PROGRAM Socket
VAR
	arSocketListen: ARRAY[1..8] OF FB_SocketListen;
	arSocketAccept: ARRAY[1..8] OF FB_SocketAccept;	
	
	arSocketConnect: ARRAY[1..8] OF FB_SocketConnect;
	arSocketReceive: ARRAY[1..8] OF FB_SocketReceive;
    arSocketSend: ARRAY[1..8] OF FB_SocketSend;	
	arSocketClose: ARRAY[1..8] OF FB_SocketClose;	
		
	arListen: ARRAY[1..8] OF BOOL;
	arhlistener: ARRAY[1..8] OF  T_HSOCKET;

	wReceiveDataBuffer: ARRAY[0..127] OF WORD;
	wSendDataBuffer: ARRAY[0..127] OF WORD;	
	
	wReceiveData: ARRAY[0..127] OF WORD;
	wSendData: ARRAY[0..127] OF WORD;
	wNullData: ARRAY[0..127] OF WORD;
	
	pbyReceiveData: ARRAY [0..255] OF BYTE;;
	pbySendData: ARRAY [0..255] OF BYTE;;
 
	byReceiveData: ARRAY [0..255] OF BYTE;;
	bySendData: ARRAY [0..255] OF BYTE;	
	
	byPrint:  ARRAY [0..MAX_STRING_LENGTH] OF BYTE;
	byPrintAuto:  ARRAY [0..MAX_STRING_LENGTH] OF BYTE;
	byPrintUser:  ARRAY [0..MAX_STRING_LENGTH] OF BYTE;
	
	iSocket: ARRAY[1..8] OF INT;
	arConnectExecute: ARRAY[1..8] OF BOOL;
	arConnectError: ARRAY[1..8] OF BOOL;
	arConnectErrId: ARRAY[1..8] OF UDINT;
	arConnectBusy: ARRAY[1..8] OF BOOL;
		
	arReceiveExecute: ARRAY[1..8] OF BOOL;
	arReceiveError: ARRAY[1..8] OF BOOL;
	arReceiveErrId: ARRAY[1..8] OF UDINT;
	arReceiveBusy: ARRAY[1..8] OF BOOL;
		
	arCloseExecute: ARRAY[1..8] OF BOOL;
	arCloseError: ARRAY[1..8] OF BOOL;
	arCloseErrId: ARRAY[1..8] OF UDINT;
	arCloseBusy: ARRAY[1..8] OF BOOL;
	arhSocket: ARRAY[1..8] OF T_HSOCKET;
	
	arSendExecute: ARRAY[1..8] OF BOOL;

	
	arSendError: ARRAY[1..8] OF BOOL;
	arSendErrId: ARRAY[1..8] OF UDINT;
	arSendBusy: ARRAY[1..8] OF BOOL;
	arTon: ARRAY [1..8] OF Ton;
	arBlink: ARRAY[1..8] OF BLINK;
	
	testString: STRING:='1';
	byteString: BYTE;
	pS: POINTER TO STRING;

	arAccept: ARRAY[1..8] OF bool;
	arListenBusy: ARRAY[1..8] OF bool;
	arAcceptBusy: ARRAY[1..8] OF bool;
	arListenError: ARRAY[1..8] OF bool;
	arAcceptError: ARRAY[1..8] OF bool;

	
	
	byPrintSend: ARRAY [0..MAX_STRING_LENGTH] OF BYTE;
	byPrintReceive: ARRAY [0..MAX_STRING_LENGTH] OF BYTE;


	iPPReceive: INT;
	diReceiveData: DINT;
	iPPSend: INT;
	iPPAccept: INT;

	
	tonFS: TON;
	
	pReceiveString: POINTER TO STRING;
	wSendCnt: WORD;
	
	
	sTestSting: STRING(255);
	arrtestBytearr: ARRAY [0..MAX_STRING_LENGTH] OF BYTE;
	arrToBytearr: ARRAY [0..MAX_STRING_LENGTH] OF BYTE;
	sToBytearrString: T_MaxString;
	sAutoPrintData: STRING(22);
	sTestPrintData: STRING(22);
	bDebugFlag: DINT;
	sTestData: STRING;
	iLen: UINT;
	rViewPrintPos: REAL;
	rPrintPosBuffer: REAL;
END_VAR

//TCP1_Client();
TCP2_Server();
pReceiveString:=ADR(pbyReceiveData);
HMI_PrinterReceiveData:=pReceiveString^;
sTestSting:=BYTEARR_TO_MAXSTRING(in:= arrtestBytearr);
arrToBytearr:=MAXSTRING_TO_BYTEARR(in:= sToBytearrString);

ACTION TCP1_Client:
(*
arSocketConnect[1](
	sSrvNetId:= , 
	sRemoteHost:= '192.168.1.199', 
	nRemotePort:= 3000, 
	bExecute:= arConnectExecute[1] , 
	tTimeout:= T#10S, 
	bBusy=> arConnectBusy[1], 
	bError=> arConnectError[1], 
	nErrId=> arConnectErrId[1], 
	hSocket=> arhSocket[1]);
		
arBlink[1](TimeH:= 1000, TimeL:= 2000, OUT=> );
	
arSocketReceive[1](
	sSrvNetId:= , 
	hSocket:=  arhSocket[1], 
	cbLen:= 255, 
	pDest:= ADR(ReceiveData[1]), 
	bExecute:= arReceiveExecute[1], 
	tTimeout:= T#1S, 
	bBusy=> arReceiveBusy[1], 
	bError=> arReceiveError[1], 
	nErrId=> arReceiveErrId[1], 
	nRecBytes=> );

arSocketSend[1](
	sSrvNetId:= , 
	hSocket:= arhSocket[1], 
	cbLen:=  255, 
	pSrc:= ADR(SendData[1]), 
	bExecute:= arSendExecute[1], 
	tTimeout:= T#1S, 
	bBusy=> arSendBusy[1], 
	bError=> arSendError[1], 
	nErrId=> arSendErrId[1]);	
	
	
arSocketClose[1](
	sSrvNetId:= , 
	hSocket:=  arhSocket[1], 
	bExecute:= arCloseExecute[1], 
	tTimeout:= T#1S, 
	bBusy=>  arCloseBusy[1], 
	bError=> arCloseError[1], 
	nErrId=> arCloseErrId[1]);



	
CASE iSocket[1] OF 
0:  
    MEMSET(destAddr:= ADR(arhSocket[1]), fillByte:= 0, n:= SIZEOF(arhSocket[1]));  
	arConnectExecute[1]:=FALSE;	
    iSocket[1]:=1;
	
1:  
	iSocket[1]:=2;
		
2:
    arConnectExecute[1]:=TRUE;	
    IF arConnectBusy[1] THEN
	   arConnectExecute[1]:=FALSE;	
       iSocket[1]:=3;
	END_IF	
	
3:  
	iSocket[1]:=4;
	
4:	
    IF arhSocket[1].handle<>0 THEN
       iSocket[1]:=10;
	ELSE IF arConnectError[1] THEN
		    iSocket[1]:=0;
		 END_IF
	END_IF


	   
10:
    arReceiveExecute[1]:=TRUE;
	iSocket[1]:=11;
	
11:
	   arReceiveExecute[1]:=FALSE;
	   iSocket[1]:=12;
12:
	IF NOT arReceiveError[1] AND NOT arReceiveBusy[1] THEN
	   iSocket[1]:=13;
	   ELSE IF arReceiveError[1] THEN
	           iSocket[1]:=90; 
            END_IF  
	END_IF 	
	
13:	
	   iSocket[1]:=20;
	
20:
	arSendExecute[1]:=TRUE; 
	iSocket[1]:=21;


21:	 
	   arSendExecute[1]:=FALSE;
	   iSocket[1]:=22;
	
22:
	IF NOT arSendError[1] AND NOT arSendBusy[1]  THEN
	   iSocket[1]:=23;
	   ELSE IF arSendError[1] THEN
	           iSocket[1]:=90;
	        END_IF
	END_IF 
       		   
23:
	   iSocket[1]:=10;


90: 
    arConnectExecute[1]:=FALSE;  
    arSendExecute[1]:=FALSE;
    arReceiveExecute[1]:=FALSE;
	arCloseExecute[1]:=TRUE;
	iSocket[1]:=91;

91: 
	   iSocket[1]:=92;

92:
	   arCloseExecute[1]:=FALSE;
	   iSocket[1]:=0;

END_CASE
*)
END_ACTION

ACTION TCP2_Server:
tonFS(IN:= TRUE, PT:= T#60S, Q=> , ET=> );

arSocketListen[2](
	sSrvNetId:= , 
	sLocalHost:= '192.168.1.10', 
	nLocalPort:= 6853, 
	bExecute:= arListen[2] OR tonFS.Q , 
	tTimeout:=, 
	bBusy=> arListenBusy[2], 
	bError=> arListenError[2], 
	nErrId=> , 
	hListener=> arhlistener[2]);
	
	
arSocketAccept[2](
	sSrvNetId:= , 
	hListener:= arhlistener[2], 
	bExecute:= arAccept[2], 
	tTimeout:= , 
	bAccepted=> , 
	bBusy=> arAcceptBusy[2], 
	bError=> arAcceptError[2], 
	nErrId=> , 
	hSocket=> arhSocket[2]);	
	
arSocketReceive[2](
	sSrvNetId:= , 
	hSocket:=  arhSocket[2], 
	cbLen:= 255, 
	pDest:= ADR(wReceiveDataBuffer), 
	bExecute:= arReceiveExecute[2], 
	tTimeout:= T#1S, 
	bBusy=> arReceiveBusy[2], 
	bError=> arReceiveError[2], 
	nErrId=> arReceiveErrId[2], 
	nRecBytes=> );

arSocketSend[2](
	sSrvNetId:= , 
	hSocket:= arhSocket[2], 
	cbLen:=  255, 
	pSrc:= ADR(wSendDataBuffer), 
	bExecute:= arSendExecute[2], 
	tTimeout:= T#1S, 
	bBusy=> arSendBusy[2], 
	bError=> arSendError[2], 
	nErrId=> arSendErrId[2]);	
	
	
arSocketClose[2](
	sSrvNetId:= , 
	hSocket:=  arhSocket[2], 
	bExecute:= arCloseExecute[2], 
	tTimeout:= T#1S, 
	bBusy=>  arCloseBusy[2], 
	bError=> arCloseError[2], 
	nErrId=> arCloseErrId[2]);	
	
	
rViewPrintPos:= arRealAxisAdmin[48].o.ActPos- rPrintPosBuffer;
	
CASE iPPAccept OF 
0:  
    MEMSET(destAddr:= ADR(wReceiveData), fillByte:= 0, n:= SIZEOF(wReceiveData));
    MEMSET(destAddr:= ADR(arhSocket[2]), fillByte:= 0, n:= SIZEOF(arhSocket[2]));  		
    iPPAccept:=1;	
1: 	
    IF arhlistener[2].handle<>0 THEN
       iPPAccept:=2;
	END_IF
2:	
	arTon[2](IN:= TRUE, PT:= T#100MS, Q=> , ET=> );	
	IF arTon[2].Q THEN
	   arTon[2](IN:= FALSE, PT:= T#100MS, Q=> , ET=> );	
	   iPPAccept:=10;
	END_IF
	   
10: arAccept[2]:=TRUE;	
    iPPAccept:=11;
	
11:
	arTon[2](IN:= TRUE, PT:= T#100MS, Q=> , ET=> );	
	IF arTon[2].Q THEN
	   arTon[2](IN:= FALSE, PT:= T#100MS, Q=> , ET=> );	
	   iPPAccept:=12;
	END_IF
	
12:	
    IF arhSocket[2].handle<>0 THEN
       iPPAccept:=20;
	   ELSE 
	   arAccept[2]:=FALSE;
	   iPPAccept:=1;
	END_IF

20:
    HMI_PrinterConnected:=TRUE;
    iPPReceive:=10;
	iPPAccept:=100;


90:  
    
    HMI_PrinterConnected:=FALSE;
	arAccept[2]:=FALSE;
    arSendExecute[2]:=FALSE;
    arReceiveExecute[2]:=FALSE;
	arCloseExecute[2]:=TRUE;
	iPPAccept:=91;

91: 
	arTon[2](IN:= TRUE, PT:= T#100MS, Q=> , ET=> );	
	IF arTon[2].Q THEN
	   arTon[2](IN:= FALSE, PT:= T#100MS, Q=> , ET=> );	
	   iPPAccept:=92;
	END_IF
	
92:
	arCloseExecute[2]:=FALSE;
	iPPAccept:=0;
END_CASE
	
CASE iPPReceive OF
	10: 
	    MEMSET(destAddr:= ADR(wReceiveDataBuffer), fillByte:= 0, n:= SIZEOF(wReceiveDataBuffer));
	    arReceiveExecute[2]:=FALSE;
		iPPReceive:=11;
		
	11:
        arTon[3](IN:= TRUE, PT:= T#100MS, Q=> , ET=> );	
		IF arTon[3].Q THEN
		   arTon[3](IN:= FALSE, PT:= T#100MS, Q=> , ET=> );	
		   iPPReceive:=20;
		END_IF
		
	20:	
	    arReceiveExecute[2]:=TRUE;
		iPPReceive:=21;
		
	21:
        arTon[3](IN:= TRUE, PT:= T#1000MS, Q=> , ET=> );	
		IF arTon[3].Q THEN
		   arTon[3](IN:= FALSE, PT:= T#1000MS, Q=> , ET=> );	
		   iPPReceive:=30;
		END_IF		
		
	30: 
        diReceiveData:=MEMCMP(pBuf1:=ADR(wReceiveDataBuffer) , pBuf2:=ADR(wNullData) , n:=SIZEOF(wNullData));
        IF 	diReceiveData<>0 THEN
		    MEMSET(destAddr:= ADR(wReceiveData), fillByte:= 0, n:= SIZEOF(wReceiveData));
		    wReceiveData:=wReceiveDataBuffer;
			pbyReceiveData[0]:=WORD_TO_BYTE(wReceiveDataBuffer[5]);
			pbyReceiveData[1]:=WORD_TO_BYTE(wReceiveDataBuffer[6]);
			pbyReceiveData[2]:=WORD_TO_BYTE(wReceiveDataBuffer[7]);
			pbyReceiveData[3]:=WORD_TO_BYTE(wReceiveDataBuffer[8]);
			pbyReceiveData[4]:=WORD_TO_BYTE(wReceiveDataBuffer[9]);
			pbyReceiveData[5]:=WORD_TO_BYTE(wReceiveDataBuffer[10]);
			pbyReceiveData[6]:=WORD_TO_BYTE(wReceiveDataBuffer[11]);
			pbyReceiveData[7]:=WORD_TO_BYTE(wReceiveDataBuffer[12]);
			pbyReceiveData[8]:=WORD_TO_BYTE(wReceiveDataBuffer[13]);
			pbyReceiveData[9]:=WORD_TO_BYTE(wReceiveDataBuffer[14]);
			pbyReceiveData[10]:=WORD_TO_BYTE(wReceiveDataBuffer[15]);
			pbyReceiveData[11]:=WORD_TO_BYTE(wReceiveDataBuffer[16]);
			pbyReceiveData[12]:=WORD_TO_BYTE(wReceiveDataBuffer[17]);
			pbyReceiveData[13]:=WORD_TO_BYTE(wReceiveDataBuffer[18]);
			pbyReceiveData[14]:=WORD_TO_BYTE(wReceiveDataBuffer[19]);
			pbyReceiveData[15]:=WORD_TO_BYTE(wReceiveDataBuffer[20]);
			pbyReceiveData[16]:=WORD_TO_BYTE(wReceiveDataBuffer[21]);
			pbyReceiveData[17]:=WORD_TO_BYTE(wReceiveDataBuffer[22]);
			pbyReceiveData[18]:=WORD_TO_BYTE(wReceiveDataBuffer[23]);
			pbyReceiveData[19]:=WORD_TO_BYTE(wReceiveDataBuffer[24]);
			pbyReceiveData[20]:=WORD_TO_BYTE(wReceiveDataBuffer[25]);
			pbyReceiveData[21]:=WORD_TO_BYTE(wReceiveDataBuffer[26]);
			pbyReceiveData[22]:=WORD_TO_BYTE(wReceiveDataBuffer[27]);			
	    END_IF
		iPPReceive:=10;
	    IF arSocketReceive[2].bError THEN
		   iPPReceive:=0;
		   iPPAccept:=90;
		END_IF
		
END_CASE

CASE iPPSend OF
	0:  IF HMI_PrinterConnected  AND glb_Un02Box.Box[HMI_PrintNo].PrintRequest AND wReceiveData[0]<>0 THEN
		   iPPSend:=10;
		ELSE IF HMI_PrinterConnected AND wReceiveData[0]<>0 AND  HMI_PrinterTest THEN
                iPPSend:=200;
			 END_IF	
	    END_IF
	10:
	   MEMSET(destAddr:= ADR(byPrintUser), fillByte:= 0, n:= SIZEOF(byPrintUser));
	   MEMSET(destAddr:= ADR(wSendDataBuffer), fillByte:= 0, n:= SIZEOF(wSendDataBuffer));
	   MEMSET(destAddr:= ADR(sAutoPrintData), fillByte:= 0, n:= SIZEOF(sAutoPrintData));
	   iLen:=INT_TO_UINT(LEN(glb_Un02Box.Box[HMI_PrintNo].PrintData));
	   MEMCPY(ADR(sAutoPrintData),ADR(glb_Un02Box.Box[HMI_PrintNo].PrintData),ilen);
	   IF NOT bDebugFlag.0 THEN
	   iPPSend:=11;
	   END_IF
	11:
	   byPrintUser:=MAXSTRING_TO_BYTEARR(sAutoPrintData);
	   IF NOT bDebugFlag.1 THEN
	   iPPSend:=20;
       END_IF
	
	   
	20:		
        wSendDataBuffer[0]:= 35;
		iPPSend:=30;
	30: 	
	    wSendCnt:=wSendCnt+1;
	    IF wSendCnt>200 THEN
		   wSendCnt:=1;
		END_IF	
		
		wSendDataBuffer[1]:=0;
		wSendDataBuffer[2]:=wSendCnt;
		wSendDataBuffer[3]:=0;
		wSendDataBuffer[4]:=44;
		wSendDataBuffer[5]:=BYTE_TO_WORD(byPrintUser[0]);
		wSendDataBuffer[6]:=BYTE_TO_WORD(byPrintUser[1]);
		wSendDataBuffer[7]:=BYTE_TO_WORD(byPrintUser[2]);
		wSendDataBuffer[8]:=BYTE_TO_WORD(byPrintUser[3]);
		wSendDataBuffer[9]:=BYTE_TO_WORD(byPrintUser[4]);
		wSendDataBuffer[10]:=BYTE_TO_WORD(byPrintUser[5]);
		wSendDataBuffer[11]:=BYTE_TO_WORD(byPrintUser[6]);
		wSendDataBuffer[12]:=BYTE_TO_WORD(byPrintUser[7]);
		wSendDataBuffer[13]:=BYTE_TO_WORD(byPrintUser[8]);
		wSendDataBuffer[14]:=BYTE_TO_WORD(byPrintUser[9]);
		wSendDataBuffer[15]:=BYTE_TO_WORD(byPrintUser[10]);
		wSendDataBuffer[16]:=BYTE_TO_WORD(byPrintUser[11]);
		wSendDataBuffer[17]:=BYTE_TO_WORD(byPrintUser[12]);
		wSendDataBuffer[18]:=BYTE_TO_WORD(byPrintUser[13]);
		wSendDataBuffer[19]:=BYTE_TO_WORD(byPrintUser[14]);
		wSendDataBuffer[20]:=BYTE_TO_WORD(byPrintUser[15]);
		wSendDataBuffer[21]:=BYTE_TO_WORD(byPrintUser[16]);
		wSendDataBuffer[22]:=BYTE_TO_WORD(byPrintUser[17]);
		wSendDataBuffer[23]:=BYTE_TO_WORD(byPrintUser[18]);
		wSendDataBuffer[24]:=BYTE_TO_WORD(byPrintUser[19]);
		wSendDataBuffer[25]:=BYTE_TO_WORD(byPrintUser[20]);
        wSendDataBuffer[26]:=BYTE_TO_WORD(byPrintUser[21]);	
		arSendExecute[2]:=FALSE;		
		iPPSend:=31;
		
		
    31:		
	    arTon[4](IN:= TRUE, PT:= T#100MS, Q=> , ET=> );	
		IF arTon[4].Q THEN
		   arTon[4](IN:= FALSE, PT:= T#100MS, Q=> , ET=> );	
		   iPPSend:=40;
		END_IF	
    40:
        arSendExecute[2]:=TRUE;
		iPPSend:=41;	
    41:
	    arTon[4](IN:= TRUE, PT:= T#10S, Q=> , ET=> );	
		IF arTon[4].Q THEN
		   arTon[4](IN:= FALSE, PT:= T#10S, Q=> , ET=> );	
		   iPPSend:=50;
		END_IF
		
	50:	
	    arTon[4](IN:= TRUE, PT:= DINT_TO_TIME(HMI_PrintMaxTime*1000), Q=> , ET=> );	
	    IF wReceiveData[2]=wSendCnt  THEN
		   arTon[4](IN:= FALSE, PT:= DINT_TO_TIME(HMI_PrintMaxTime*1000), Q=> , ET=> );
		   iPPSend:=60;
		   ELSE IF arTon[4].Q THEN
				   arTon[4](IN:= FALSE, PT:= DINT_TO_TIME(HMI_PrintMaxTime*1000), Q=> , ET=> );
				   iPPSend:=51;
		   END_IF
		END_IF
    51: 
	    HMI_PrinterFault:=TRUE;
	    iPPSend:=52;
	52: IF NOT HMI_PrinterFault THEN
		   iPPSend:=60;
	    END_IF
    60:
	
	    glb_Un02Box.Box[HMI_PrintNo].PrintRequest:= FALSE;
		arSendExecute[2]:=FALSE;
	    iPPSend:=0;	

		
	200: 
		MEMSET(destAddr:= ADR(byPrint), fillByte:= 0, n:= SIZEOF(byPrint));
		MEMSET(destAddr:= ADR(wSendDataBuffer), fillByte:= 0, n:= SIZEOF(wSendDataBuffer));
	    MEMSET(destAddr:= ADR(sTestPrintData), fillByte:= 0, n:= SIZEOF(sTestPrintData));
	    iLen:=INT_TO_UINT(LEN(HMI_PrinterTestData));
	    MEMCPY(ADR(sTestPrintData),ADR(HMI_PrinterTestData),ilen);		
	    byPrint:=MAXSTRING_TO_BYTEARR(sTestPrintData);	
		
		iPPSend:=210;	
		
    210:
		wSendDataBuffer[0]:= 35;
		iPPSend:=220;
		
	220:	
	    wSendCnt:=wSendCnt+1;
	    IF wSendCnt>200 THEN
		   wSendCnt:=1;
		END_IF
	
		wSendDataBuffer[1]:=0;
		wSendDataBuffer[2]:=wSendCnt;
		wSendDataBuffer[3]:=0;
		wSendDataBuffer[4]:=44;
		wSendDataBuffer[5]:=BYTE_TO_WORD(byPrint[0]);
		wSendDataBuffer[6]:=BYTE_TO_WORD(byPrint[1]);
		wSendDataBuffer[7]:=BYTE_TO_WORD(byPrint[2]);
		wSendDataBuffer[8]:=BYTE_TO_WORD(byPrint[3]);
		wSendDataBuffer[9]:=BYTE_TO_WORD(byPrint[4]);
		wSendDataBuffer[10]:=BYTE_TO_WORD(byPrint[5]);
		wSendDataBuffer[11]:=BYTE_TO_WORD(byPrint[6]);
		wSendDataBuffer[12]:=BYTE_TO_WORD(byPrint[7]);
		wSendDataBuffer[13]:=BYTE_TO_WORD(byPrint[8]);
		wSendDataBuffer[14]:=BYTE_TO_WORD(byPrint[9]);
		wSendDataBuffer[15]:=BYTE_TO_WORD(byPrint[10]);
		wSendDataBuffer[16]:=BYTE_TO_WORD(byPrint[11]);
		wSendDataBuffer[17]:=BYTE_TO_WORD(byPrint[12]);
		wSendDataBuffer[18]:=BYTE_TO_WORD(byPrint[13]);
		wSendDataBuffer[19]:=BYTE_TO_WORD(byPrint[14]);
		wSendDataBuffer[20]:=BYTE_TO_WORD(byPrint[15]);
		wSendDataBuffer[21]:=BYTE_TO_WORD(byPrint[16]);
		wSendDataBuffer[22]:=BYTE_TO_WORD(byPrint[17]);
		wSendDataBuffer[23]:=BYTE_TO_WORD(byPrint[18]);
		wSendDataBuffer[24]:=BYTE_TO_WORD(byPrint[19]);
		wSendDataBuffer[25]:=BYTE_TO_WORD(byPrint[20]);
        wSendDataBuffer[26]:=BYTE_TO_WORD(byPrint[21]);

		
		arSendExecute[2]:=FALSE;
		iPPSend:=221;
		
    221:		
	    arTon[4](IN:= TRUE, PT:= T#1000MS, Q=> , ET=> );	
		IF arTon[4].Q THEN
		   arTon[4](IN:= FALSE, PT:= T#1000MS, Q=> , ET=> );	
		   iPPSend:=230;
		END_IF	
    230:
        arSendExecute[2]:=TRUE;
		iPPSend:=231;			

    231:
	    arTon[4](IN:= TRUE, PT:= T#1000MS, Q=> , ET=> );	
		IF arTon[4].Q THEN
		   arTon[4](IN:= FALSE, PT:= T#1000MS, Q=> , ET=> );	
		   iPPSend:=240;
		END_IF
		
	240:
	    arTon[4](IN:= TRUE, PT:= DINT_TO_TIME(HMI_PrintMaxTime*1000), Q=> , ET=> );	
	    IF wReceiveData[2]=wSendCnt  THEN
		   arTon[4](IN:= FALSE, PT:= DINT_TO_TIME(HMI_PrintMaxTime*1000), Q=> , ET=> );
		   iPPSend:=0; 
		   arSendExecute[2]:=FALSE;
		   ELSE IF arTon[4].Q THEN
			    arTon[4](IN:= FALSE, PT:= DINT_TO_TIME(HMI_PrintMaxTime*1000), Q=> , ET=> );
				iPPSend:=241;
		   END_IF	   
		END_IF		
		
		
	241: HMI_PrinterFault:=TRUE;
	     arSendExecute[2]:=FALSE;
         iPPSend:=0;	
		
END_CASE
END_ACTION

END_PROGRAM

(* stored: Version 1.1.0.1, ProductVersion 3.1.4024.6
   POU Socket: Id {7e84310f-93f3-4b07-a568-04fd6b0a1c40}, SpecialFunc None
   Action TCP1_Client: Id {878c632a-644b-496b-a0b0-e840ef3f30b4}
   Action TCP2_Server: Id {96dbe25d-dcf9-4b64-aeb7-adfecb578df0} *)
